FUNCTION_BLOCK E_F_TRIG (* Composite Function Block Type *)
  (* Standard: 61499-2 *)
  (* Version 0.0, 9/9/2026, lizar, Schneider Electric, template *)
  PACKAGE Main;
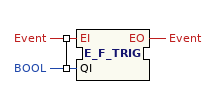
  EVENT_INPUT
    EI WITH QI; (* Initialization Request *)
  END_EVENT
  EVENT_OUTPUT
    EO; (* Initialization Confirm *)
  END_EVENT
  VAR_INPUT
    QI : BOOL; (* Input event qualifier *)
  END_VAR
  FBS
    FB1 : E_D_FF;
    FB2 : E_PERMIT;
    FB3 : NOT_42C76073DCEB1A7A; {SET_ATTRIBUTE(Configuration.GenericFBType.InterfaceParams, Runtime.Standard#CNT:=1;OUT${CNT$}:BOOL)}
  END_FBS
  EVENT_CONNECTIONS
    EI TO FB1.CLK;
    FB1.EO TO FB3.REQ;
    FB3.CNF TO FB2.EI;
    FB2.EO TO EO;
  END_CONNECTIONS
  DATA_CONNECTIONS
    QI TO FB1.D;
    FB1.Q TO FB3.IN1;
    FB3.OUT1 TO FB2.PERMIT;
  END_CONNECTIONS
END_FUNCTION_BLOCK
